FUNCTION_BLOCK PidController
VAR
	desiredValue_ : LREAL;
	actualValue_ : LREAL;
	previousValue_ : LREAL;
	error_ : LREAL;
	controlOutput_ : LREAL;
	
	cycleTime_ : UDINT;
	
	firstLoop_ : BOOL := TRUE;
	
	kp_ : LREAL;
	ki_ : LREAL;
	kd_ : LREAL;
	
	p_ : LREAL;
	i_ : LREAL;
	d_ : LREAL;
END_VAR


METHOD calculateDifferential

d_ := kd_ * ((actualValue_ - previousValue_) / cycleTime_);

IF previousValue_ = 0 THEN
	d_ := 0;
END_IF

previousValue_ := actualValue_;
END_METHOD


METHOD calculateIntegral

i_ := i_ + ki_ * error_;
END_METHOD


METHOD calculateOutput : LREAL

calculateOutput := p_ + i_ + d_;
END_METHOD


METHOD calculateProportional

p_ := kp_ * error_;
END_METHOD


METHOD cyclic
VAR_INPUT
	actualValue : LREAL;
END_VAR
VAR_OUTPUT
	controlOutput : LREAL;
END_VAR

IF firstLoop_ THEN
	getCycleTime();
	firstLoop_ := FALSE;
END_IF

actualValue_ := actualValue;
error_ := desiredValue_ - actualValue_;

// P
calculateProportional();
// I
calculateIntegral();
// D 
calculateProportional();

controlOutput := calculateOutput();
END_METHOD

//FB_Init is always available implicitly and it is used primarily for initialization.
//The return value is not evaluated. For a specific influence, you can also declare the
//methods explicitly and provide additional code there with the standard initialization
//code. You can evaluate the return value.
METHOD FB_Init: BOOL
VAR_INPUT
    bInitRetains: BOOL; // TRUE: the retain variables are initialized (reset warm / reset cold)
    bInCopyCode: BOOL;  // TRUE: the instance will be copied to the copy code afterward (online change)
		desiredValue : LREAL;
		kp : LREAL;
		ki : LREAL;
		kd : LREAL;
END_VAR

desiredValue_ := desiredValue;
kp_ := kp;
ki_ := ki;
kd_ := kd;
END_METHOD


METHOD getCycleTime
VAR
	taskIndex : DINT;
END_VAR

taskIndex := Tc2_System.GETCURTASKINDEXEX();
IF taskIndex > 0 THEN
    cycleTime_ := TwinCAT_SystemInfoVarList._TaskInfo[taskIndex].CycleTime;
END_IF
END_METHOD


METHOD reset

actualValue_ := 0;
previousValue_ := 0;
error_ := 0;
controlOutput_ := 0;
cycleTime_ := 0;
firstLoop_ := TRUE;
p_ := 0;
i_ := 0;
d_ := 0;
END_METHOD

END_FUNCTION_BLOCK

(* stored: Version 1.1.0.1, ProductVersion 3.1.4026.6
   POU PidController: Id {f0fe1ff9-cf00-4079-8b85-73b781bbb7df}, SpecialFunc None
   Method calculateDifferential: Id {d72610e8-b849-4d78-b7e6-a0a51a0546da}
   Method calculateIntegral: Id {ae3494a9-c3f3-421a-ac47-f814e80fb549}
   Method calculateOutput: Id {46507d54-ada6-4753-bd5f-c6033668a7b4}
   Method calculateProportional: Id {f128500b-6413-4df5-a8dc-0dffe3cf25ce}
   Method cyclic: Id {df297eb9-d813-4b4c-98f1-3a28fa58764e}
   Method FB_Init: Id {9a068693-6288-4318-89c6-345ec40ca419}
   Method getCycleTime: Id {25083f72-f29f-459d-b5cd-a7a6c0986574}
   Method reset: Id {8101f034-77b4-4451-92e5-1e7a94b8c87c} *)
